FUNCTION_BLOCK EtherCatMaster
VAR_GENERIC CONSTANT
	FRAMES	   : UINT := 1;
	SYNC_UNITS : UINT := 2;
END_VAR
EXTENDS CyclicComponent IMPLEMENTS I_EtherCatMasterDiagnostic, I_Initializable, I_TaskResult, I_Simulatable, I_CoeTransferScheduler
VAR
	EcMaster	AT %I*	: ST_EtherCatMasterInfo;
	FrmXWcState AT %I*	: ARRAY[0..(FRAMES - 1)] OF WORD;
	ConfiguredSlaveInfo : ARRAY[0..MAX_EC_SLAVES] OF ST_EcSlaveConfigData;
	SlavesState			: ARRAY[0..MAX_EC_SLAVES] OF ST_EcExtendedSlaveState;
	SlaveTopologyInfo	: ARRAY[0..MAX_EC_SLAVES] OF ST_TopologyDataEx;
	// Configured slave index + 1 by (EtherCAT address - FIRST_SLAVE_ADDR); 0 = no slave at that address
	AddrToIndex			: ARRAY[0..MAX_EC_SLAVES] OF UINT;
	SyncUnit			: ARRAY[0..(SYNC_UNITS - 1)] OF SyncUnitTask('Sync Unit', THIS^, ConfiguredSlaveInfo, SlaveTopologyInfo);
	IoDevice			: ARRAY[0..MAX_EC_SLAVES] OF EtherCatIoDevice('Io Device');
	// CoE transfers in flight - only these are serviced each cycle (I_CoeTransferScheduler)
	ActiveCoe			: ARRAY[0..MAX_EC_SLAVES] OF I_CoeTransfer;
	ActiveCoeCount		: UINT;
	EventProvider		: I_EtherCatDiagnosticEventProvider;
END_VAR

VAR
	InitSequenceState								 : UDINT;
	SlaveSequence									 : UDINT;
	RunSlaveDiag, LastFramesWcStatesOk				 : BOOL;
	LastChangeCount, LastSlaveCount, LastMasterState : UINT;
	EcStartupCycles									 : UINT;
	SlaveCountUsed									 : UINT;  // configured slaves covered by the arrays, latched in Initialize
	ScanIndex										 : UINT;  // slave position of the running multi-cycle pass
	SyncUnitScan									 : UINT;  // sync unit of the running assignment pass
	FirstDiagIndex									 : UINT;  // first slave that is not OP or reports a link problem
	AnyDiag											 : BOOL;
	SyncUnitsAssigned								 : BOOL;
	WaitCycles										 : UDINT; // ADS watchdog of the running wait step
	GetConfiguredSlaves								 : FB_EcGetConfSlaves;
	GetMasterFrameCount								 : FB_EcMasterFrameCount;
	GetAllSlaveStates								 : FB_EcGetAllExtSlaveStates;
	GetSlaveTopologyInfo							 : FB_EcGetSlaveTopologyInfo;
END_VAR

VAR
	{attribute 'hide'}
	_Initialized : BOOL;
	{attribute 'hide'}
	_Error : BOOL;
	{attribute 'hide'}
	_Busy : BOOL;
	{attribute 'hide'}
	_ErrorId : UDINT;
	{attribute 'hide'}
	_ErrorSource : E_EcErrorSource;
	{attribute 'hide'}
	_Simulated : BOOL;
	{attribute 'hide'}
	Config : ST_EcSlaveConfigData;
	{attribute 'hide'}
	State : ST_EcExtendedSlaveState;
	{attribute 'hide'}
	NullIoDevice : EtherCatIoDevice('NullIoDevice') := (Configuration := Config, State := State);
	{attribute 'hide'}
	_LocalAmsNetId : T_AmsNetId;
	{attribute 'hide'}
	_MasterAmsNetId : T_AmsNetId;
END_VAR

VAR CONSTANT
	FIRST_SLAVE_ADDR  : UINT  := 1001;	 // TwinCAT assigns EtherCAT addresses from 1001 in configuration order
	ADS_TIMEOUT		  : TIME  := T#5S;
	ERROR_ADS_TIMEOUT : UDINT := 16#745; // ADS client: timeout elapsed (watchdog abort)
END_VAR

// Counts the cycles of the running wait step; TRUE once MaxCycles is exceeded.
METHOD PRIVATE AdsWatchdogExpired : BOOL
VAR_INPUT
	MaxCycles : UDINT;
END_VAR
WaitCycles		   := WaitCycles + 1;
AdsWatchdogExpired := WaitCycles > MaxCycles;
END_METHOD

// Rebuilds the address map from the configured slaves (SlaveCountUsed entries).
METHOD PROTECTED BuildAddrToIndex
VAR
	i : UINT;
END_VAR
MEMSET(ADR(AddrToIndex), 0, SIZEOF(AddrToIndex));

i := 0;
WHILE i < SlaveCountUsed DO
	MapSlaveAddress(i);
	i := i + 1;
END_WHILE
END_METHOD

// TRUE while a diagnostic sequence runs. A pass over n slaves takes up to n / SLAVES_PER_CYCLE cycles,
// so Error/ErrorId of a change land that many cycles after the trigger.
{attribute 'monitoring' := 'call'}
PROPERTY Busy : BOOL
GET
Busy := _Busy;
END_GET
END_PROPERTY

{attribute 'monitoring' := 'call'}
PROPERTY ConfiguredSlaveCount : UINT
GET
ConfiguredSlaveCount := EcMaster.CfgSlaveCount;
END_GET
END_PROPERTY

METHOD CyclicLogic
VAR
	i : UINT;
END_VAR
IF NOT Initialized THEN
	Initialize();
	RETURN;
END_IF

IF Simulated THEN
	_Busy		 := FALSE;
	_Error		 := FALSE;
	_ErrorId	 := 0;
	_ErrorSource := E_EcErrorSource.None;
ELSE
	IF NOT _Busy THEN
		IF (LastChangeCount <> EcMaster.ChangeCount) THEN
			RunSlaveDiag := TRUE;
		ELSIF ((EcMaster.CfgSlaveCount <> EcMaster.SlaveCount) AND (LastSlaveCount <> EcMaster.SlaveCount)) THEN
			RunSlaveDiag := TRUE;
		ELSIF FramesWcStatesOk() <> LastFramesWcStatesOk THEN
			RunSlaveDiag := TRUE;
		END_IF

		IF RunSlaveDiag THEN
			LastChangeCount		 := EcMaster.ChangeCount;
			LastSlaveCount		 := EcMaster.SlaveCount;
			LastFramesWcStatesOk := FramesWcStatesOk();
		END_IF
	END_IF

	MasterState();
	SlaveState();
	FOR i := 0 TO (SYNC_UNITS - 1) DO
		SyncUnit[i].CyclicLogic();
	END_FOR

	_Busy := SlaveSequence <> 0;
END_IF

(* Only CoE transfers in flight are serviced; idle io devices cost nothing per cycle. *)
ServiceCoeTransfers();
END_METHOD

// Leaves the slave evaluation: assigns the sync units once they resolved their slave lists, otherwise idles.
METHOD PRIVATE EndDiagnosticPass
IF NOT SyncUnitsAssigned AND_THEN SyncUnitsResolved() THEN
	SyncUnitScan  := 0;
	ScanIndex	  := 0;
	SlaveSequence := 40;
ELSE
	SlaveSequence := 0;
END_IF
END_METHOD

{attribute 'monitoring' := 'call'}
PROPERTY Error : BOOL
GET
Error := _Error;
END_GET
END_PROPERTY

// Raw code of ErrorSource: DevState word (Master), slave index (Slave), ADS error id (Ads), step (Sequence).
{attribute 'monitoring' := 'call'}
PROPERTY ErrorId : UDINT
GET
ErrorId := _ErrorId;
END_GET
END_PROPERTY

{attribute 'monitoring' := 'call'}
PROPERTY ErrorSource : E_EcErrorSource
GET
ErrorSource := _ErrorSource;
END_GET
END_PROPERTY

// Raises the slave events for one configured slave. TRUE when a fault was latched (Error, ErrorSource.Slave).
METHOD PROTECTED EvaluateSlave : BOOL
VAR_INPUT
	Index : UINT;
END_VAR

VAR
	DiagByte : BYTE;
END_VAR
IF SlaveTopologyInfo[Index].nStatusBits.4 THEN
	RETURN; // member of a hot connect group: absence or a non-OP state is not a fault
END_IF

DiagByte := SlavesState[Index].deviceState AND 16#0F;
IF DiagByte <> EC_DEVICE_STATE_OP THEN
	IF SlavesState[Index].deviceState.7 THEN // slave is disabled - warning only
		IF EventProvider <> 0 THEN
			EventProvider.RaiseEtherCatDiagnosticEvent(E_EtherCatMaster.SlaveDisabled, ConfiguredSlaveInfo[Index].sName);
		END_IF
	ELSE
		IF EventProvider <> 0 THEN
			EventProvider.RaiseEtherCatDiagnosticEvent(E_EtherCatMaster.SlaveError, ConfiguredSlaveInfo[Index].sName, LookupSlaveState(Index));
		END_IF

		SetError(E_EcErrorSource.Slave, Index);
		EvaluateSlave := TRUE;
		RETURN;
	END_IF
END_IF

DiagByte := SlavesState[Index].linkState AND 16#0F;
IF DiagByte <> EC_LINK_STATE_OK THEN
	IF EventProvider <> 0 THEN
		EventProvider.RaiseEtherCatDiagnosticEvent(E_EtherCatMaster.SlaveError, ConfiguredSlaveInfo[Index].sName, LookupSlaveState(Index));
	END_IF

	SetError(E_EcErrorSource.Slave, Index);
	EvaluateSlave := TRUE;
END_IF
END_METHOD

// Latches the error, logs Message and parks the init sequence in step 999.
METHOD PRIVATE FailInit
VAR_INPUT
	Source	: E_EcErrorSource;
	ErrorId : UDINT;
	Message : T_MaxString;
END_VAR
SetError(Source, ErrorId);
Trace.LogMessage(Name, Message);
InitSequenceState := 999;
END_METHOD

// Latches the error and aborts the running diagnostic sequence.
METHOD PRIVATE FailSequence
VAR_INPUT
	Source	: E_EcErrorSource;
	ErrorId : UDINT;
END_VAR
SetError(Source, ErrorId);
SlaveSequence := 0;
END_METHOD

(*FB_Init is always available implicitly and it is used primarily for initialization.
The return value is not evaluated. For a specific influence, you can also declare the
methods explicitly and provide additional code there with the standard initialization
code. You can evaluate the return value.*)
METHOD FB_Init : BOOL
VAR_INPUT
	(* TRUE: the retain variables are initialized (reset warm / reset cold)*)
	bInitRetains : BOOL;

	(* TRUE: the instance will be copied to the copy code afterward (online change)   *)
	bInCopyCode		: BOOL;
	Name			: T_MaxString;
	EcStartupCycles : UINT;
END_VAR
THIS^.EcStartupCycles := EcStartupCycles;
END_METHOD

METHOD PROTECTED FramesWcStatesOk : BOOL
VAR
	i : UDINT;
END_VAR
FramesWcStatesOk := TRUE;
IF GetMasterFrameCount.nFrames = 0 THEN
	RETURN;
END_IF

FOR i := 0 TO (MIN(GetMasterFrameCount.nFrames, FRAMES) - 1) DO
	IF FrmXWcState[i] <> 0 THEN
		FramesWcStatesOk := FALSE;
		EXIT;
	END_IF
END_FOR
END_METHOD

// O(1) through the address map. Returns the null device (and logs a warning) for unknown addresses.
METHOD GetIoDeviceByAddr : I_EcIoDevice
VAR_INPUT
	Addr : WORD;
END_VAR

VAR
	Idx : DINT;
END_VAR
IF NOT Initialized THEN
	GetIoDeviceByAddr := NullIoDevice;
	RETURN;
END_IF

Idx := GetSlaveIndexByAddr(WORD_TO_UINT(Addr));
IF Idx >= 0 THEN
	GetIoDeviceByAddr := IoDevice[Idx];
ELSE
	Trace.LogMessage(Name, CONCAT('GetIoDeviceByAddr: no configured slave at address ', TO_STRING(WORD_TO_UINT(Addr))));
	GetIoDeviceByAddr := NullIoDevice;
END_IF
END_METHOD

// Linear search over the configured slaves: call once and keep the result.
// Returns the null device (and logs a warning) if no slave carries that name.
METHOD GetIoDeviceByName : I_EcIoDevice
VAR_INPUT
	Name : STRING(31);
END_VAR

VAR
	i : UINT;
END_VAR
IF NOT Initialized THEN
	GetIoDeviceByName := NullIoDevice;
	RETURN;
END_IF

i := 0;
WHILE i < SlaveCountUsed DO
	IF IoDevice[i].Name = Name THEN
		GetIoDeviceByName := IoDevice[i];
		RETURN;
	END_IF
	i := i + 1;
END_WHILE

Trace.LogMessage(THIS^.Name, CONCAT('GetIoDeviceByName: no configured slave named ', Name));
GetIoDeviceByName := NullIoDevice;
END_METHOD

// Configured slave index (0-based) of the slave with EtherCAT address Addr, -1 if none.
// O(1) for the dense range FIRST_SLAVE_ADDR .. FIRST_SLAVE_ADDR + MAX_EC_SLAVES, linear search otherwise.
METHOD GetSlaveIndexByAddr : DINT
VAR_INPUT
	Addr : UINT;
END_VAR

VAR
	i : UINT;
END_VAR
GetSlaveIndexByAddr := -1;

IF (Addr >= FIRST_SLAVE_ADDR) AND_THEN ((Addr - FIRST_SLAVE_ADDR) <= MAX_EC_SLAVES) THEN
	IF AddrToIndex[Addr - FIRST_SLAVE_ADDR] <> 0 THEN
		GetSlaveIndexByAddr := AddrToIndex[Addr - FIRST_SLAVE_ADDR] - 1;
	END_IF
	RETURN; // the map is complete for this range
END_IF

(* Addresses outside the dense range (assigned by the user): linear search. *)
i := 0;
WHILE i < SlaveCountUsed DO
	IF ConfiguredSlaveInfo[i].nAddr = Addr THEN
		GetSlaveIndexByAddr := i;
		RETURN;
	END_IF
	i := i + 1;
END_WHILE
END_METHOD

// Init sequence: local AMS Net ID (0) - configured slaves (10) - topology (20) - frame count (30) -
// sync units (40) - startup cycles, io device wiring and address map (50). Step 999 = failed, see trace.
METHOD Initialize
VAR_INST
	GetLocalAmsNetId : FB_GetLocalAmsNetId;
	StartCycles		 : UINT;
END_VAR

VAR
	i : UDINT;
	k : UINT;
END_VAR
IF NOT _Error AND NOT Simulated THEN
	IF F_GetMappingStatus(ADR(EcMaster.AmsNetID), SIZEOF(EcMaster.AmsNetID)) = EplcMappingStatus.MS_Unmapped THEN
		FailInit(E_EcErrorSource.Sequence, InitSequenceState, 'Init Failed - EcMaster.AmsNetID not mapped to the EtherCAT master!');
	ELSIF F_GetMappingStatus(ADR(EcMaster.DevID), SIZEOF(EcMaster.DevID)) = EplcMappingStatus.MS_Unmapped THEN
		FailInit(E_EcErrorSource.Sequence, InitSequenceState, 'Init Failed - EcMaster.DevID not mapped to the EtherCAT master!');
	ELSIF F_GetMappingStatus(ADR(EcMaster.DevState), SIZEOF(EcMaster.DevState)) = EplcMappingStatus.MS_Unmapped THEN
		FailInit(E_EcErrorSource.Sequence, InitSequenceState, 'Init Failed - EcMaster.DevState not mapped to the EtherCAT master!');
	ELSIF F_GetMappingStatus(ADR(EcMaster.ChangeCount), SIZEOF(EcMaster.ChangeCount)) = EplcMappingStatus.MS_Unmapped THEN
		FailInit(E_EcErrorSource.Sequence, InitSequenceState, 'Init Failed - EcMaster.ChangeCount not mapped to the EtherCAT master!');
	ELSIF F_GetMappingStatus(ADR(EcMaster.SlaveCount), SIZEOF(EcMaster.SlaveCount)) = EplcMappingStatus.MS_Unmapped THEN
		FailInit(E_EcErrorSource.Sequence, InitSequenceState, 'Init Failed - EcMaster.SlaveCount not mapped to the EtherCAT master!');
	ELSIF F_GetMappingStatus(ADR(EcMaster.CfgSlaveCount), SIZEOF(EcMaster.CfgSlaveCount)) = EplcMappingStatus.MS_Unmapped THEN
		FailInit(E_EcErrorSource.Sequence, InitSequenceState, 'Init Failed - EcMaster.CfgSlaveCount not mapped to the EtherCAT master!');
	END_IF
END_IF

IF _Error THEN
	RETURN;
END_IF

IF Simulated THEN
	FOR i := 0 TO (SYNC_UNITS - 1) DO
		SyncUnit[i].EventProvider := EventProvider;
		SyncUnit[i].Simulated	  := Simulated;
		SyncUnit[i].Initialize();
		IF NOT SyncUnit[i].Initialized THEN
			RETURN;
		END_IF
	END_FOR

	_Initialized := TRUE;
	RETURN;
END_IF

GetLocalAmsNetId(tTimeOut := T#1S);
_MasterAmsNetId := F_CreateAmsNetId(EcMaster.AmsNetID);
GetMasterFrameCount(sNetId := _MasterAmsNetId, tTimeout := ADS_TIMEOUT);
GetConfiguredSlaves(sNetId				:= _MasterAmsNetId,
					pArrEcConfSlaveInfo := ADR(ConfiguredSlaveInfo),
					cbBufLen			:= SlaveCountUsed * SIZEOF(ConfiguredSlaveInfo[0]),
					tTimeout			:= ADS_TIMEOUT);
GetSlaveTopologyInfo(sNetId	  := _MasterAmsNetId,
					 pAddrBuf := ADR(SlaveTopologyInfo),
					 cbBufLen := TopologyBufLen(),
					 tTimeout := ADS_TIMEOUT);

CASE InitSequenceState OF
	0: (* local AMS Net ID *)
		GetLocalAmsNetId.bExecute := TRUE;
		WaitCycles				  := 0;
		NextMinorStep(InitSequenceState);

	1:
		IF GetLocalAmsNetId.bBusy THEN
			IF AdsWatchdogExpired(ADS_WAIT_CYCLES) THEN
				GetLocalAmsNetId.bExecute := FALSE;
				FailInit(E_EcErrorSource.Ads, ERROR_ADS_TIMEOUT, 'Init Failed - GetLocalAmsNetId timed out!');
			END_IF
		ELSIF GetLocalAmsNetId.bError THEN
			GetLocalAmsNetId.bExecute := FALSE;
			FailInit(E_EcErrorSource.Ads, GetLocalAmsNetId.nErrId, 'Init Failed - GetLocalAmsNetId!');
		ELSE
			GetLocalAmsNetId.bExecute := FALSE;
			_LocalAmsNetId			  := GetLocalAmsNetId.AddrString;
			WaitCycles				  := 0;
			NextStep(InitSequenceState);
		END_IF

	10: (* configured slaves, read sized to the configured count *)
		IF EcMaster.CfgSlaveCount = 0 THEN
			IF AdsWatchdogExpired(ADS_WAIT_CYCLES) THEN
				FailInit(E_EcErrorSource.Sequence, InitSequenceState, 'Init Failed - EcMaster.CfgSlaveCount stays 0: no slaves configured or EcMaster not linked!');
			END_IF
			RETURN;
		END_IF

		IF EcMaster.CfgSlaveCount > (MAX_EC_SLAVES + 1) THEN
			FailInit(E_EcErrorSource.Sequence, EcMaster.CfgSlaveCount, 'Init Failed - more slaves configured than EtherCatParameter.MAX_EC_SLAVES + 1 can hold!');
			RETURN;
		END_IF

		SlaveCountUsed				 := EcMaster.CfgSlaveCount;
		GetConfiguredSlaves.bExecute := TRUE;
		WaitCycles					 := 0;
		NextMinorStep(InitSequenceState);

	11:
		IF GetConfiguredSlaves.bBusy THEN
			IF AdsWatchdogExpired(INIT_WAIT_CYCLES) THEN
				GetConfiguredSlaves.bExecute := FALSE;
				FailInit(E_EcErrorSource.Ads, ERROR_ADS_TIMEOUT, 'Init Failed - reading the configured EtherCAT slaves timed out!');
			END_IF
		ELSIF GetConfiguredSlaves.bError THEN
			GetConfiguredSlaves.bExecute := FALSE;
			FailInit(E_EcErrorSource.Ads, GetConfiguredSlaves.nErrorId, 'Init Failed - configured EtherCAT slaves could not be read - check linking of the EtherCAT master FB!');
		ELSE
			GetConfiguredSlaves.bExecute := FALSE;
			WaitCycles					 := 0;
			NextStep(InitSequenceState);
		END_IF

	20: (* topology: the hot connect flags are needed by the slave evaluation and the sync units *)
		GetSlaveTopologyInfo.bExecute := TRUE;
		WaitCycles					  := 0;
		NextMinorStep(InitSequenceState);

	21:
		IF GetSlaveTopologyInfo.bBusy THEN
			IF AdsWatchdogExpired(INIT_WAIT_CYCLES) THEN
				GetSlaveTopologyInfo.bExecute := FALSE;
				FailInit(E_EcErrorSource.Ads, ERROR_ADS_TIMEOUT, 'Init Failed - reading the EtherCAT topology timed out!');
			END_IF
		ELSIF GetSlaveTopologyInfo.bError THEN
			GetSlaveTopologyInfo.bExecute := FALSE;
			FailInit(E_EcErrorSource.Ads, GetSlaveTopologyInfo.nErrId, 'Init Failed - EtherCAT topology could not be read!');
		ELSE
			GetSlaveTopologyInfo.bExecute := FALSE;
			WaitCycles					  := 0;
			NextStep(InitSequenceState);
		END_IF

	30: (* frame count *)
		GetMasterFrameCount.bExecute := TRUE;
		WaitCycles					 := 0;
		NextMinorStep(InitSequenceState);

	31:
		IF GetMasterFrameCount.bBusy THEN
			IF AdsWatchdogExpired(ADS_WAIT_CYCLES) THEN
				GetMasterFrameCount.bExecute := FALSE;
				FailInit(E_EcErrorSource.Ads, ERROR_ADS_TIMEOUT, 'Init Failed - reading the EtherCAT frame count timed out!');
			END_IF
		ELSIF GetMasterFrameCount.bError THEN
			GetMasterFrameCount.bExecute := FALSE;
			FailInit(E_EcErrorSource.Ads, GetMasterFrameCount.nErrId, 'Init Failed - configured EtherCAT frames could not be read!');
		ELSE
			GetMasterFrameCount.bExecute := FALSE;
			IF GetMasterFrameCount.nFrames = 0 THEN
				FailInit(E_EcErrorSource.Sequence, InitSequenceState, 'Init Failed - the EtherCAT master reports no cyclic frames!');
				RETURN;
			END_IF

			IF GetMasterFrameCount.nFrames > FRAMES THEN
				FailInit(E_EcErrorSource.Sequence, GetMasterFrameCount.nFrames, 'Init Failed - increase the FRAMES generic parameter and link FrmXWcState[x] to the master!');
				RETURN;
			END_IF

			FOR i := 0 TO (GetMasterFrameCount.nFrames - 1) DO
				IF F_GetMappingStatus(ADR(FrmXWcState[i]), SIZEOF(FrmXWcState[i])) = EplcMappingStatus.MS_Unmapped THEN
					FailInit(E_EcErrorSource.Sequence, i, 'Init Failed - FrmXWcState[x] not mapped to the EtherCAT master!');
					RETURN;
				END_IF
			END_FOR

			NextStep(InitSequenceState);
		END_IF

	40: (* sync units *)
		FOR i := 0 TO (SYNC_UNITS - 1) DO
			SyncUnit[i].EventProvider := EventProvider;
			SyncUnit[i].Initialize();
			IF SyncUnit[i].Error THEN
				FailInit(E_EcErrorSource.Sequence, i, 'Init Failed - a sync unit could not be initialised (see its trace message)!');
				RETURN;
			END_IF

			IF NOT SyncUnit[i].Initialized THEN
				RETURN;
			END_IF
		END_FOR

		NextStep(InitSequenceState);

	50: (* let the master settle, then build the address map *)
		StartCycles := StartCycles + 1;
		IF StartCycles >= EcStartupCycles THEN
			BuildAddrToIndex();
			ScanIndex := 0;
			NextMinorStep(InitSequenceState);
		END_IF

	51: (* wire the io devices, SLAVES_PER_CYCLE per cycle *)
		FOR k := 1 TO SLAVES_PER_CYCLE DO
			IF ScanIndex >= SlaveCountUsed THEN
				EXIT;
			END_IF

			IoDevice[ScanIndex].AmsNetId	  := EcMaster.AmsNetID;
			IoDevice[ScanIndex].Name		  := ConfiguredSlaveInfo[ScanIndex].sName;
			IoDevice[ScanIndex].State		  REF= SlavesState[ScanIndex];
			IoDevice[ScanIndex].Configuration REF= ConfiguredSlaveInfo[ScanIndex];
			IoDevice[ScanIndex].CoeScheduler  := THIS^;
			ScanIndex						  := ScanIndex + 1;
		END_FOR

		IF ScanIndex >= SlaveCountUsed THEN
			_Initialized := TRUE;
		END_IF

	999: (* Fail - look at the trace message in the ADS log *)
END_CASE
END_METHOD

{attribute 'monitoring' := 'call'}
PROPERTY Initialized : BOOL
GET
Initialized := _Initialized;
END_GET
SET
_Initialized := Initialized;
END_SET
END_PROPERTY

{attribute 'monitoring' := 'call'}
PROPERTY LocalAmsNetId : T_AmsNetId
GET
LocalAmsNetId := _LocalAmsNetId;
END_GET
END_PROPERTY

METHOD PROTECTED LookupMasterState : STRING
VAR_INPUT
	State : UINT;
END_VAR
IF State.0 THEN
	LookupMasterState := 'Link error';
ELSIF State.1 THEN
	LookupMasterState := 'I/O locked after link error (I/O reset required)';
ELSIF State.2 THEN
	LookupMasterState := 'Link error (redundancy adapter)';
ELSIF State.3 THEN
	LookupMasterState := 'Missing one frame (redundancy mode)';
ELSIF State.4 THEN
	LookupMasterState := 'Out of send resources (I/O reset required)';
ELSIF State.5 THEN
	LookupMasterState := 'Watchdog triggered';
ELSIF State.6 THEN
	LookupMasterState := 'Ethernet driver (miniport) NOT found';
ELSIF State.7 THEN
	LookupMasterState := 'I/O reset active';
ELSIF State.8 THEN
	LookupMasterState := 'At least one device in INIT state';
ELSIF State.9 THEN
	LookupMasterState := 'At least one device in PRE-OP state';
ELSIF State.10 THEN
	LookupMasterState := 'At least one device in SAFE-OP state';
ELSIF State.11 THEN
	LookupMasterState := 'At least one device indicates an error state';
ELSIF State.12 THEN
	LookupMasterState := 'DC not in sync';
ELSE
	LookupMasterState := 'State not found';
END_IF
END_METHOD

METHOD PROTECTED LookupSlaveState : STRING
VAR_INPUT
	Slave : UINT;
END_VAR

VAR_INST
	DiagByte	: BYTE;
	BitMaskDiag : BYTE := 16#0F;
END_VAR
(* State *)
BitMaskDiag := 16#0F;
DiagByte	:= SlavesState[Slave].deviceState AND BitMaskDiag;
CASE DiagByte OF
	EC_DEVICE_STATE_INIT:
		LookupSlaveState := 'Init';

	EC_DEVICE_STATE_PREOP:
		LookupSlaveState := 'Pre-op';

	EC_DEVICE_STATE_BOOTSTRAP:
		LookupSlaveState := 'Boot';

	EC_DEVICE_STATE_SAFEOP:
		LookupSlaveState := 'Safe-op';

	EC_DEVICE_STATE_OP:
		LookupSlaveState := 'OP';

ELSE
	LookupSlaveState := '';
END_CASE

(* Additional State Bits *)
IF SlavesState[Slave].deviceState.4 THEN // EC_DEVICE_STATE_ERROR
	LookupSlaveState := CONCAT(LookupSlaveState, ' - ');
	LookupSlaveState := CONCAT(LookupSlaveState, 'State machine error in the EtherCAT slave');
END_IF

IF SlavesState[Slave].deviceState.5 THEN // EC_DEVICE_STATE_INVALID_VPRS
	LookupSlaveState := CONCAT(LookupSlaveState, ' - ');
	LookupSlaveState := CONCAT(LookupSlaveState, 'Invalid vendor ID');
END_IF

IF SlavesState[Slave].deviceState.6 THEN // EC_DEVICE_STATE_INITCMD_ERROR
	LookupSlaveState := CONCAT(LookupSlaveState, ' - ');
	LookupSlaveState := CONCAT(LookupSlaveState, 'Error during sending of initialization commands');
END_IF

IF SlavesState[Slave].deviceState.7 THEN // EC_DEVICE_STATE_DISABLED
	LookupSlaveState := CONCAT(LookupSlaveState, ' - ');
	LookupSlaveState := CONCAT(LookupSlaveState, 'Slave is disabled');
END_IF

//_____________________________________________________________________________________________________

(* Link States *)
IF SlavesState[Slave].linkState.0 THEN // EC_LINK_STATE_NOT_PRESENT
	LookupSlaveState := CONCAT(LookupSlaveState, ' - ');
	LookupSlaveState := CONCAT(LookupSlaveState, 'No EtherCAT communication with the EtherCAT slave');
END_IF

IF SlavesState[Slave].linkState.1 THEN // EC_LINK_STATE_LINK_WITHOUT_COMM
	LookupSlaveState := CONCAT(LookupSlaveState, ' - ');
	LookupSlaveState := CONCAT(LookupSlaveState, 'Error AT port X');
END_IF

IF SlavesState[Slave].linkState.2 THEN // EC_LINK_STATE_MISSING_LINK
	LookupSlaveState := CONCAT(LookupSlaveState, ' - ');
	LookupSlaveState := CONCAT(LookupSlaveState, 'Missing link AT port X');
END_IF

IF SlavesState[Slave].linkState.3 THEN // EC_LINK_STATE_ADDITIONAL_LINK
	LookupSlaveState := CONCAT(LookupSlaveState, ' - ');
	LookupSlaveState := CONCAT(LookupSlaveState, 'Additional link AT port X');
END_IF

(* Additional State Bits *)
IF SlavesState[Slave].linkState.4 THEN // EC_LINK_STATE_PORT_A
	LookupSlaveState := CONCAT(LookupSlaveState, ' - ');
	LookupSlaveState := CONCAT(LookupSlaveState, 'Port 0');
END_IF

IF SlavesState[Slave].linkState.5 THEN // EC_LINK_STATE_PORT_B
	LookupSlaveState := CONCAT(LookupSlaveState, ' - ');
	LookupSlaveState := CONCAT(LookupSlaveState, 'Port 1');
END_IF

IF SlavesState[Slave].linkState.6 THEN // EC_LINK_STATE_PORT_C
	LookupSlaveState := CONCAT(LookupSlaveState, ' - ');
	LookupSlaveState := CONCAT(LookupSlaveState, 'Port 2');
END_IF

IF SlavesState[Slave].linkState.7 THEN // EC_LINK_STATE_PORT_D
	LookupSlaveState := CONCAT(LookupSlaveState, ' - ');
	LookupSlaveState := CONCAT(LookupSlaveState, 'Port 3');
END_IF
END_METHOD

// Enters the configured slave Index into the address map if its address lies in the dense range.
METHOD PROTECTED MapSlaveAddress
VAR_INPUT
	Index : UINT;
END_VAR

VAR
	Addr : UINT;
END_VAR
Addr := ConfiguredSlaveInfo[Index].nAddr;
IF (Addr >= FIRST_SLAVE_ADDR) AND_THEN ((Addr - FIRST_SLAVE_ADDR) <= MAX_EC_SLAVES) THEN
	AddrToIndex[Addr - FIRST_SLAVE_ADDR] := Index + 1;
END_IF
END_METHOD

{attribute 'monitoring' := 'call'}
PROPERTY MasterAmsNetId : T_AmsNetId
GET
MasterAmsNetId := _MasterAmsNetId;
END_GET
END_PROPERTY

// Raises one MasterError event per DevState change while slaves are missing. TRUE when an error was latched.
METHOD PROTECTED MasterState : BOOL
VAR_INPUT
END_VAR
IF LastMasterState = EcMaster.DevState THEN
	RETURN;
END_IF

LastMasterState := EcMaster.DevState;

IF (EcMaster.DevState <> 0) AND (EcMaster.SlaveCount < EcMaster.CfgSlaveCount) THEN
	IF EventProvider <> 0 THEN
		EventProvider.RaiseEtherCatDiagnosticEvent(E_EtherCatMaster.MasterError, LookupMasterState(EcMaster.DevState));
	END_IF

	SetError(E_EcErrorSource.Master, EcMaster.DevState);
	MasterState := TRUE;
END_IF
END_METHOD

// I_CoeTransferScheduler: adds a CoE transfer to the set serviced by CyclicLogic (idempotent).
METHOD Register : BOOL
VAR_INPUT
	Transfer : I_CoeTransfer;
END_VAR

VAR
	i : UINT;
END_VAR
IF Transfer = 0 THEN
	RETURN;
END_IF

i := 0;
WHILE i < ActiveCoeCount DO
	IF ActiveCoe[i] = Transfer THEN
		Register := TRUE;
		RETURN;
	END_IF
	i := i + 1;
END_WHILE

IF ActiveCoeCount > MAX_EC_SLAVES THEN
	RETURN; // full
END_IF

ActiveCoe[ActiveCoeCount] := Transfer;
ActiveCoeCount			  := ActiveCoeCount + 1;
Register				  := TRUE;
END_METHOD

METHOD RegisterEventProvider
VAR_INPUT
	EventProvider : I_EtherCatDiagnosticEventProvider;
END_VAR
THIS^.EventProvider := EventProvider;
END_METHOD

METHOD Reset
IF EventProvider <> 0 THEN
	EventProvider.Reset();
END_IF

LastMasterState				  := 0;
LastChangeCount				  := 0;
LastSlaveCount				  := 0;
LastFramesWcStatesOk		  := FALSE;
_Error						  := FALSE;
_ErrorId					  := 0;
_ErrorSource				  := E_EcErrorSource.None;
SlaveSequence				  := 0;
RunSlaveDiag				  := FALSE;
GetAllSlaveStates.bExecute	  := FALSE;
GetSlaveTopologyInfo.bExecute := FALSE;
END_METHOD

// Calls CyclicLogic of every registered CoE transfer and drops the ones that finished.
METHOD PRIVATE ServiceCoeTransfers
VAR
	i : UINT;
END_VAR
i := 0;
WHILE i < ActiveCoeCount DO
	ActiveCoe[i].CyclicLogic();
	IF ActiveCoe[i].Busy THEN
		i := i + 1;
	ELSE
		(* finished: move the last entry into the gap and service it in this cycle as well *)
		ActiveCoeCount			  := ActiveCoeCount - 1;
		ActiveCoe[i]			  := ActiveCoe[ActiveCoeCount];
		ActiveCoe[ActiveCoeCount] := 0;
	END_IF
END_WHILE
END_METHOD

METHOD PROTECTED SetError
VAR_INPUT
	Source	: E_EcErrorSource;
	ErrorId : UDINT;
END_VAR
_Error		 := TRUE;
_ErrorSource := Source;
_ErrorId	 := ErrorId;
END_METHOD

{attribute 'monitoring' := 'call'}
PROPERTY Simulated : BOOL
GET
Simulated := _Simulated;
END_GET
SET
_Simulated := Simulated;
END_SET
END_PROPERTY

{attribute 'monitoring' := 'call'}
PROPERTY SlaveCount : UINT
GET
SlaveCount := EcMaster.SlaveCount;
END_GET
END_PROPERTY

// TRUE if the slave is not in OP with a clean link (any state or link bit set).
METHOD PROTECTED SlaveNeedsDiagnostic : BOOL
VAR_INPUT
	Index : UINT;
END_VAR
SlaveNeedsDiagnostic := (SlavesState[Index].deviceState <> EC_DEVICE_STATE_OP) OR (SlavesState[Index].linkState <> 0);
END_METHOD

// Slave diagnostic sequence, run on every trigger (ChangeCount, slave count, frame WC state):
//  10/11 read all slave states (sized to the configured count)
//  12    classify, SLAVES_PER_CYCLE slaves per cycle; a clean network ends here
//  20/21 read the topology (hot connect flags) - only when a slave needs a diagnostic
//  30    evaluate from the first suspicious slave, stop at the first fault
//  40    assign the sync unit of every slave, once, after the sync units resolved their lists
METHOD PROTECTED SlaveState : BOOL
VAR
	k	: UINT;
	Idx : DINT;
END_VAR
GetSlaveTopologyInfo(sNetId	  := _MasterAmsNetId,
					 pAddrBuf := ADR(SlaveTopologyInfo),
					 cbBufLen := TopologyBufLen(),
					 tTimeout := ADS_TIMEOUT);

GetAllSlaveStates(sNetId	:= _MasterAmsNetId,
				  pStateBuf := ADR(SlavesState),
				  cbBufLen	:= SlaveCountUsed * SIZEOF(SlavesState[0]),
				  tTimeout	:= ADS_TIMEOUT);

CASE SlaveSequence OF
	(* Wait for a trigger *)
	0:
		IF RunSlaveDiag THEN
			RunSlaveDiag  := FALSE;
			SlaveSequence := 10;
		ELSIF NOT SyncUnitsAssigned AND_THEN SyncUnitsResolved() THEN
			EndDiagnosticPass();
		END_IF

	(* Read slave states *)
	10:
		GetAllSlaveStates.bExecute := TRUE;
		WaitCycles				   := 0;
		NextMinorStep(SlaveSequence);

	11:
		IF GetAllSlaveStates.bBusy THEN
			IF AdsWatchdogExpired(ADS_WAIT_CYCLES) THEN
				GetAllSlaveStates.bExecute := FALSE;
				FailSequence(E_EcErrorSource.Ads, ERROR_ADS_TIMEOUT);
			END_IF
		ELSIF GetAllSlaveStates.bError THEN
			GetAllSlaveStates.bExecute := FALSE;
			FailSequence(E_EcErrorSource.Ads, GetAllSlaveStates.nErrId);
		ELSE
			GetAllSlaveStates.bExecute := FALSE;
			ScanIndex				   := 0;
			AnyDiag					   := FALSE;
			FirstDiagIndex			   := 0;
			NextMinorStep(SlaveSequence);
		END_IF

	(* Classify: find the first slave that needs a diagnostic *)
	12:
		FOR k := 1 TO SLAVES_PER_CYCLE DO
			IF ScanIndex >= SlaveCountUsed THEN
				EXIT;
			END_IF

			IF SlaveNeedsDiagnostic(ScanIndex) THEN
				AnyDiag		   := TRUE;
				FirstDiagIndex := ScanIndex;
				EXIT;
			END_IF

			ScanIndex := ScanIndex + 1;
		END_FOR

		IF AnyDiag THEN
			SlaveSequence := 20;
		ELSIF ScanIndex >= SlaveCountUsed THEN
			EndDiagnosticPass(); // every slave OP with a clean link: no topology read, no evaluation
		END_IF

	(* Update topology *)
	20:
		GetSlaveTopologyInfo.bExecute := TRUE;
		WaitCycles					  := 0;
		NextMinorStep(SlaveSequence);

	21:
		IF GetSlaveTopologyInfo.bBusy THEN
			IF AdsWatchdogExpired(ADS_WAIT_CYCLES) THEN
				GetSlaveTopologyInfo.bExecute := FALSE;
				FailSequence(E_EcErrorSource.Ads, ERROR_ADS_TIMEOUT);
			END_IF
		ELSIF GetSlaveTopologyInfo.bError THEN
			GetSlaveTopologyInfo.bExecute := FALSE;
			FailSequence(E_EcErrorSource.Ads, GetSlaveTopologyInfo.nErrId);
		ELSE
			GetSlaveTopologyInfo.bExecute := FALSE;
			ScanIndex					  := FirstDiagIndex;
			SlaveSequence				  := 30;
		END_IF

	(* Evaluate slave errors from the first suspicious slave on *)
	30:
		FOR k := 1 TO SLAVES_PER_CYCLE DO
			IF ScanIndex >= SlaveCountUsed THEN
				EXIT;
			END_IF

			IF EvaluateSlave(ScanIndex) THEN
				ScanIndex := SlaveCountUsed; // fault latched: stop the pass
				EXIT;
			END_IF

			ScanIndex := ScanIndex + 1;
		END_FOR

		IF ScanIndex >= SlaveCountUsed THEN
			EndDiagnosticPass();
		END_IF

	(* Assign the sync unit of every slave (once) *)
	40:
		FOR k := 1 TO SLAVES_PER_CYCLE DO
			IF SyncUnitScan >= SYNC_UNITS THEN
				EXIT;
			END_IF

			IF ScanIndex >= SyncUnit[SyncUnitScan].SlaveCount THEN
				SyncUnitScan := SyncUnitScan + 1;
				ScanIndex	 := 0;
			ELSE
				Idx := GetSlaveIndexByAddr(SyncUnit[SyncUnitScan].SlaveAddress(ScanIndex));
				IF Idx >= 0 THEN
					IoDevice[Idx].SyncUnit := SyncUnit[SyncUnitScan];
				END_IF

				ScanIndex := ScanIndex + 1;
			END_IF
		END_FOR

		IF SyncUnitScan >= SYNC_UNITS THEN
			SyncUnitsAssigned := TRUE;
			SlaveSequence	  := 0;
		END_IF

ELSE
	(* Sequence error: unknown step *)
	FailSequence(E_EcErrorSource.Sequence, SlaveSequence);
END_CASE
END_METHOD

// TRUE once every sync unit has read and resolved its slave list.
METHOD PRIVATE SyncUnitsResolved : BOOL
VAR
	i : UINT;
END_VAR
SyncUnitsResolved := TRUE;
FOR i := 0 TO (SYNC_UNITS - 1) DO
	IF NOT SyncUnit[i].SlavesResolved THEN
		SyncUnitsResolved := FALSE;
		RETURN;
	END_IF
END_FOR
END_METHOD

// Byte length of the topology read: one entry per configured slave, not the whole array.
METHOD PRIVATE TopologyBufLen : UDINT
TopologyBufLen := SlaveCountUsed * SIZEOF(SlaveTopologyInfo[0]);
END_METHOD

END_FUNCTION_BLOCK

(* stored: Version 1.1.0.1, ProductVersion 3.1.4026.21
   POU EtherCatMaster: Id {e9f0f328-f6e9-478d-a143-06ac013b96e0}, SpecialFunc None
   Folder _Internal: Id {ca0b50fd-5048-4aec-b945-6ade741b5cc3}
   Folder CoE: Id {3a013ee2-7997-4313-a622-78d410a5c6d2}
   Folder Diagnostic: Id {8daf5ba7-ec56-4aa2-87f5-e02cf302f316}
   Folder Initialize: Id {70d62c55-9a6e-4608-a13a-af986e41c0cf}
   Folder Resettable: Id {3af3d3da-4a00-45c9-a31e-fe08287c134d}
   Folder TaskResult: Id {8aae4edb-d4d6-4720-af63-e947524eb0f2}
   Method AdsWatchdogExpired: Id {3b9bd3d5-6590-4dd4-868c-f84365f0df38}
   Method BuildAddrToIndex: Id {540611c4-ced8-4f68-9d63-bc81cccaef12}
   Property Busy: Id {a8d6e216-d136-48f1-a6ee-beda6d975c86}
   Get Get: Id {4056a01c-0c87-4417-bd5a-9b0e2daa64f5}
   Property ConfiguredSlaveCount: Id {fad5d2d6-9a3e-0291-3bce-eb8536172a8c}
   Get Get: Id {62ec34ab-2a7d-0373-052b-2643e3f7533b}
   Method CyclicLogic: Id {78fc609d-40b9-4518-b70e-60c3ef93632e}
   Method EndDiagnosticPass: Id {a2e8164c-889e-4970-853b-1e9658378f69}
   Property Error: Id {fd2aad37-acbd-4549-8dff-3cc1e8b69d66}
   Get Get: Id {80679826-41d5-4b2a-92e4-bce3af7fb62b}
   Property ErrorId: Id {76e2677e-85b8-4192-ae01-7f29edcaffcd}
   Get Get: Id {c59f189e-2b3d-447d-8383-1ed95dba4997}
   Property ErrorSource: Id {17e49a29-0c1e-4905-860e-026e3ec8b8ce}
   Get Get: Id {f9b69b38-90d1-403e-a932-a7fc61f6b82a}
   Method EvaluateSlave: Id {9023d524-15b7-4b34-acbc-4468eb23bb1b}
   Method FailInit: Id {4984ebc0-ef47-45e8-a10b-3591d1da83e0}
   Method FailSequence: Id {7dc00690-6d23-4b1f-ab9e-e84f63f4ef5b}
   Method FB_Init: Id {b13f5ee7-b35d-4d18-9795-7f71c11f59d6}
   Method FramesWcStatesOk: Id {d8515602-a931-0646-062f-139b29a44aad}
   Method GetIoDeviceByAddr: Id {8fec52b1-8c69-4759-b15f-16e0bfdd0031}
   Method GetIoDeviceByName: Id {13f2fd00-8fca-4d64-97a3-0bb868e7b598}
   Method GetSlaveIndexByAddr: Id {49de51a0-75fa-43d3-9637-c84ac886b692}
   Method Initialize: Id {59fc31be-2fef-4308-9217-c3cfb6c18f0b}
   Property Initialized: Id {462f1142-9a6c-459f-809a-d563cfeef048}
   Get Get: Id {b67dbeea-ed7d-4fcb-ad02-e417a2e86968}
   Set Set: Id {93d7895b-12f1-47ef-9db9-da3095578fb1}
   Property LocalAmsNetId: Id {a970c90e-4636-418a-85de-aa121c8437d5}
   Get Get: Id {428487ba-9f27-4d2c-9f0f-2d1d34923b7b}
   Method LookupMasterState: Id {77909b3a-0ac2-4bf6-a988-7eb95f542820}
   Method LookupSlaveState: Id {2b979181-e45f-4339-bf02-a4112dadec98}
   Method MapSlaveAddress: Id {375c31cd-934d-4614-b398-2e47ba3ae9b0}
   Property MasterAmsNetId: Id {e8191ac3-4bf6-4260-9bd6-73f87a18d477}
   Get Get: Id {cd0137ef-9d12-42f0-957e-c261bf7bfde0}
   Method MasterState: Id {9cab473b-cce9-4d54-aadc-9cb8f27d7c22}
   Method Register: Id {af1bba30-9816-4532-9ef4-ab7b63e9c3b6}
   Method RegisterEventProvider: Id {3c83d169-3fdc-4962-9915-fa3129e33709}
   Method Reset: Id {ee94ff59-f1a9-498f-aa45-98618a0c1c63}
   Method ServiceCoeTransfers: Id {05356306-57eb-4767-8dbb-3b6da6cd102b}
   Method SetError: Id {54454f9e-58e9-4682-b57f-abdd8c767e72}
   Property Simulated: Id {aa6d861b-93bc-45a2-853a-7b9fd1cc7e49}
   Get Get: Id {cc7febd7-07c6-461f-ab58-a79f9f2f810a}
   Set Set: Id {6f7e37d4-83d8-4e75-a97b-cc1689d77fd4}
   Property SlaveCount: Id {bfc36d0d-748f-4330-826a-e7f9a3550123}
   Get Get: Id {8ba43fb2-7af8-4a46-9c1a-f74e5d772835}
   Method SlaveNeedsDiagnostic: Id {bab5ddbf-5759-4fc8-9d73-93879e28cb5f}
   Method SlaveState: Id {483b8cf5-1244-4799-bded-62d3800d6efa}
   Method SyncUnitsResolved: Id {5054c0c0-c40a-449a-95f1-194f3792089a}
   Method TopologyBufLen: Id {2a906241-c190-4ecd-8467-1699bf9f6338} *)
